FUNCTION_BLOCK fbV2_MainStationProcess

(*************************************************************** Ver.B1 - fbV2_StnSeqProcess - 161101 **************************************************************]

 	- Add 'bEffTimePriorityEn' to cutoff the process once effective time reached.																	
	- Change naming from 'bProcessCompleteBasedMasterTime' to 'bMinMaxEn'. 
	- 	
	- 
[****************************************************************************************************************************************************************************************************)

VAR_INPUT
	(*fbStnSeqProcess*)
	bAutoStartPbEn									: BOOL;
	bSavePB_Uni 									: BOOL; 														(*Universal*) (* Input - HMI - Save Push Button on Touchscreen*)
	bLoadPB_Uni 									: BOOL;														(*Universal*) (* Input - HMI - Load Push Button on Touchscreen*)
	bClearPB_SSER									: BOOL;
	bClearPB_SSUR									: BOOL;
	bTrackerEn										: BOOL;														(*During Tracker, it will only call arm when process completed*)
	bTrackerBasedOnPreviousTime					: BOOL;
	bMinMaxEn(*bProcessCompleteBasedMasterTime*)		: BOOL;
	bEffTimePriorityEn									: BOOL;
	bBasketTransferCallArmInterlock			: BOOL; (* Temporary -> for GPM Only*)

	(*fbGnrStationMasterController*)
	iCurrentStationAddress_Fix 							: INT;															(*Individual*) (* Input - Define current station no so that this fb know which array number to used*)
	iPreCallArmTime_Uni								: INT;															(*Universal*) (* Input - Pre-Call Arm Time, Program will call arm if the Total process timeEV Equal or Lesser than this value*)
	ARbAlternateStnEn								: ARRAY [1..iAlternateSetQty] OF BOOL;
	AR2siAlternateStn 									: ARRAY [1..iAlternateSetQty, 1..iAlternateStnQty] OF INT;

	
	
END_VAR

VAR_IN_OUT PERSISTENT

	(*fbStnSeqProcess*)
(*	DsStnSeqProInput_Ind 						: DS_StnSeqProInput;												(*Individual*) (* Input - PV of Instrument (Temperature, pressure, vacuum and etc), Signal of Sensor to allowed program under the current station status.*)
*)	DSStnSeqProcessCtrl_Ind			 		: DS_fbStnSeqProcessCtrl;											(*Individual*) (* InOut - Link with fbStnSeqProcess, so that this fb know the full status of fbStnSeqProcess and determine which action to take*)

	DsStnSeqRepStore_Ind 					: DSV2_fbStationSequenceRecipeStore; 								(*Individual*) (* InOut - HMI - The full set of DataStructure-StationSequenceRecipe should selectively display on HMI so that user can customise the recipe by choosing/configure the parameters.*)
	DsStnSubRepStore_Ind 					: DS_fbStationSubRecipeStore; 										(*Individual*) (* InOut - HMI - The full set of DataStructure-StationSubRecipe should selectively display on HMI so that user can customise the recipe by choosing/configure the parameters.*)
	DsStnSeqRepCall_Ind 						: DSV2_fbStationSequenceRecipeCall;									(*Individual*) (* InOut - Used to call StationSequenceRecipe Detail from fbStationSequenceRecipe*)
	DsStnSubRepCall_Ind 						: DS_fbStationSubRecipeCall;										(*Individual*) (* InOut - Used to call StationSubRecipe Detail from fbStationSubRecipe*)
	ARDsSSERSourceMinMaxTime_Uni						: ARRAY [1..iStnQty] OF DSV2_SSERSourceMinMaxTime;

	(*fbGnrStationMasterController*)
	ARbProductRecipeCallEn_Uni 				: ARRAY [0..iStnQty] OF BOOL;										(*Universal*) (* Output - Link with fbGnrProductRecipeMemory, Array based on Current Station No, the fbGnrProductRecipeMemory will start Read info from Memory when this bool turn on*)
	ARiProductRecipeNoCall_Uni 				: ARRAY [0..iStnQty] OF INT;										(*Universal*) (* Output - Link with fbGnrProductRecipeMemory, Array based on Current Station No, the read out from fbGnrProductRecipeMemory is based on this Product Recipe No*)
	ARiProductRecipeStepCall_Uni 				: ARRAY [0..iStnQty] OF INT;										(*Universal*) (* Output - Link with fbGnrProductRecipeMemory, Array based on Current Station No, the read out from fbGnrProductRecipeMemory is based on this Product Recipe Step No*)

	DSfbGnrProductRecipeMemoryOut_Uni 		: DSV2_fbGnrProductRecipeMemoryOut;								(*Universal*) (* Input - Link with fbGnrProductRecipeMemory, all the read out info from fbGnrProductRecipeMemory will store in this DataStucture*)

	ARbArmReady_Uni						: ARRAY [1..iArmQty] OF BOOL;										(* Universal*) (* Input  - From ArmPnpFB, This signal is used to confirm if the arm is ready and idling*)

	ARiStnNoToCalledArm_Uni					: ARRAY [0..iArmQty] OF INT; 										(*Universal*) (* Output - Link with fbArmPnP, Array based on Arm No, The Int will store which Station that calling the Arm*)
	ARDSGnrFeedArmPnpParameter_Uni		: ARRAY [0..iArmQty] OF DSV2_Gnr_CalledArmPnpParameter; 			(*Universal*) (* Output - Link with fbArmPnP, Array based on Current Station No, Arm should move based on this DataStructure Info*)

	ARDSLdBasketInfo_Uni		 			: ARRAY [0..iLdStnQty] OF DSV2_BasketInfo;								(*Input - Loading CONFIRM Basket Info*)
	ARDSUldBasketInfo_Uni		 			: ARRAY [0..iUldStnQty] OF DSV2_BasketInfo;							(*Input - Uloading CONFIRM Basket Info*)
	ARDsStnBasketInfo_Uni					: ARRAY [0..iStnQty] OF DSV2_BasketInfo;								(*Input - Station Basket Info*)



END_VAR

VAR_OUTPUT PERSISTENT
	bSaveInd_Uni 								: BOOL; 														(*Universal*) (* Output - HMI - Save Indicator on Touchscreen*)
	bLoadInd_Uni 								: BOOL; 														(*Universal*) (* Output - HMI - Load Indicator on Touchscreen*)
	bClearInd_SSER 								: BOOL;
	bClearInd_SSUR 								: BOOL;
(*	DSStnSeqProOutput_Ind 						:DS_StnSeqProOutput;											(*Individual*) (* Output - To Control Output - When process running, instrument should control by the output in this Data structure*)
*)

	bStationProcessCompleted : BOOL;
END_VAR



VAR PERSISTENT
	(*fbStnSeqProcess*)
	StnSeqProcessfb						: fbV2_StnSeqProcess;
	bStnSeqProcessStartInterlock			: BOOL;																	(*Individual*) (* Input - Interlocking to Enable the StnSeqProcess Start Signal, It might used on those station with Sliding door for close confirmation before process start*)

	(*fbGnrStationMasterController*)
	GnrStationMasterControllerfb				: fbV2_GnrStationMasterController;
	bStnSeqProcessSt						: BOOL;																(* Output - Link with fbStnSeqProcess, After Read out from fbGnrProductRecipeMemory, this fb will trigger this Bool to start the StnSeqProcess*)
	DSGnrBufferCalledArmPnpParameter 		: DSV2_Gnr_CalledArmPnpParameter;									(* Internal used, Buffer Data Structure read out from fbGnrProductRecipeMemory*)
	DSGnrBuffersPnpSequenceDescription		: STRING (99);														(* Internal used, Buffer Description read out from fbGnrProductRecipeMemory*)
	ARiPreviousStnSeqTotalProcessTime 		: ARRAY [0..iProductRecipeArrayQty] OF INT;								(* Internal used, Previous Total Process Time will save into this Array, Array based on StationSequenceNo*)
	iCallStep									: INT;																(* Internal used, to monitor the current Step so that you can indentify the error of this function block if stucked*)
	DSBasketInfo_Ind 							: DSV2_BasketInfo;														(*Individual*) (* InOut - Basket Information that comes into current station*)
	iNonStopCurrentProcessTime: INT;
END_VAR
VAR
	bLdStnConfirm: BOOL;
	bUldStnConfirm: BOOL;
	bStn1Confirm: BOOL;
	bGreaterStn1Confirm: BOOL;
	bLesserStnQtyConfirm: BOOL;
	bEqualStnQtyConfirm: BOOL;
	iTotalProcessTimeSV: INT;
	fbV2BasketInfoFinder_Ind: fbV2_BasketInfoFinder;
	iTotalProcessTimeCallForGnrStationMC: INT;
	iMasterTimeCallArmCountDownTime: INT;
	iMasterTimeBasedProcessCompleteFlag : BOOL;


	iMasterTimeBasedProcessCompleteFlagHR: BOOL;
	iProductRecipeBuffer: INT;
	bProductRecipeNoChangedFlag: BOOL;
END_VAR
VAR // added by the converter: edge detectors and wires of the graphical bodies
    _w1, _w2 : INT;
END_VAR

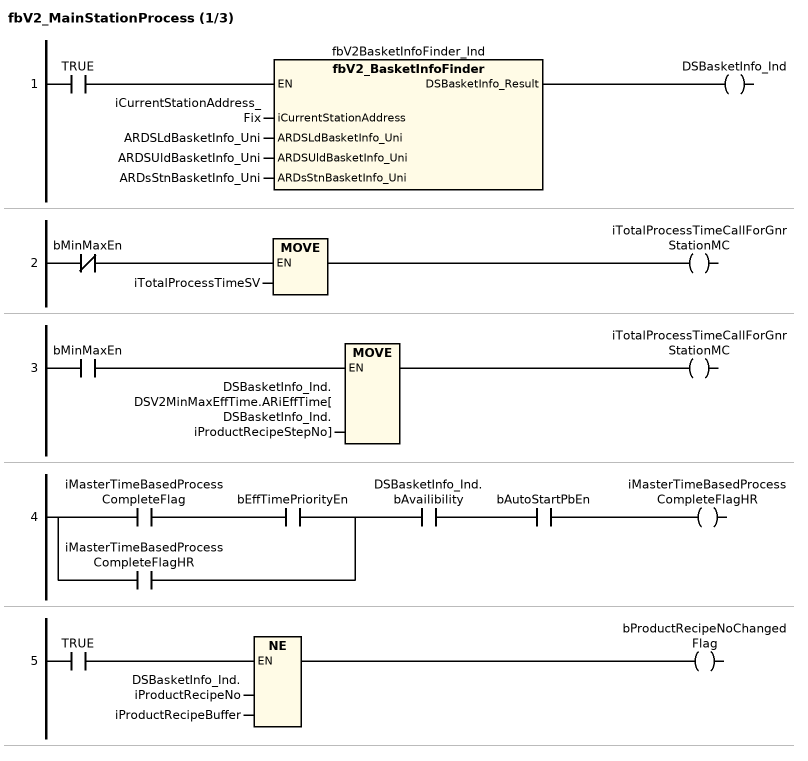
// NETWORK 1
fbV2BasketInfoFinder_Ind(
    iCurrentStationAddress := iCurrentStationAddress_Fix,
    ARDSLdBasketInfo_Uni := ARDSLdBasketInfo_Uni,
    ARDSUldBasketInfo_Uni := ARDSUldBasketInfo_Uni,
    ARDsStnBasketInfo_Uni := ARDsStnBasketInfo_Uni); // fbV2_BasketInfoFinder
DSBasketInfo_Ind := fbV2BasketInfoFinder_Ind.DSBasketInfo_Result;

// NETWORK 2
IF NOT bMinMaxEn THEN _w1 := iTotalProcessTimeSV; END_IF
iTotalProcessTimeCallForGnrStationMC := _w1;

// NETWORK 3
IF bMinMaxEn THEN
    _w2 := DSBasketInfo_Ind.DSV2MinMaxEffTime.ARiEffTime[DSBasketInfo_Ind.iProductRecipeStepNo];
END_IF
iTotalProcessTimeCallForGnrStationMC := _w2;

// NETWORK 4
iMasterTimeBasedProcessCompleteFlagHR := (iMasterTimeBasedProcessCompleteFlag AND bEffTimePriorityEn OR iMasterTimeBasedProcessCompleteFlagHR) AND DSBasketInfo_Ind.bAvailibility AND bAutoStartPbEn;

// NETWORK 5
bProductRecipeNoChangedFlag := DSBasketInfo_Ind.iProductRecipeNo <> iProductRecipeBuffer;

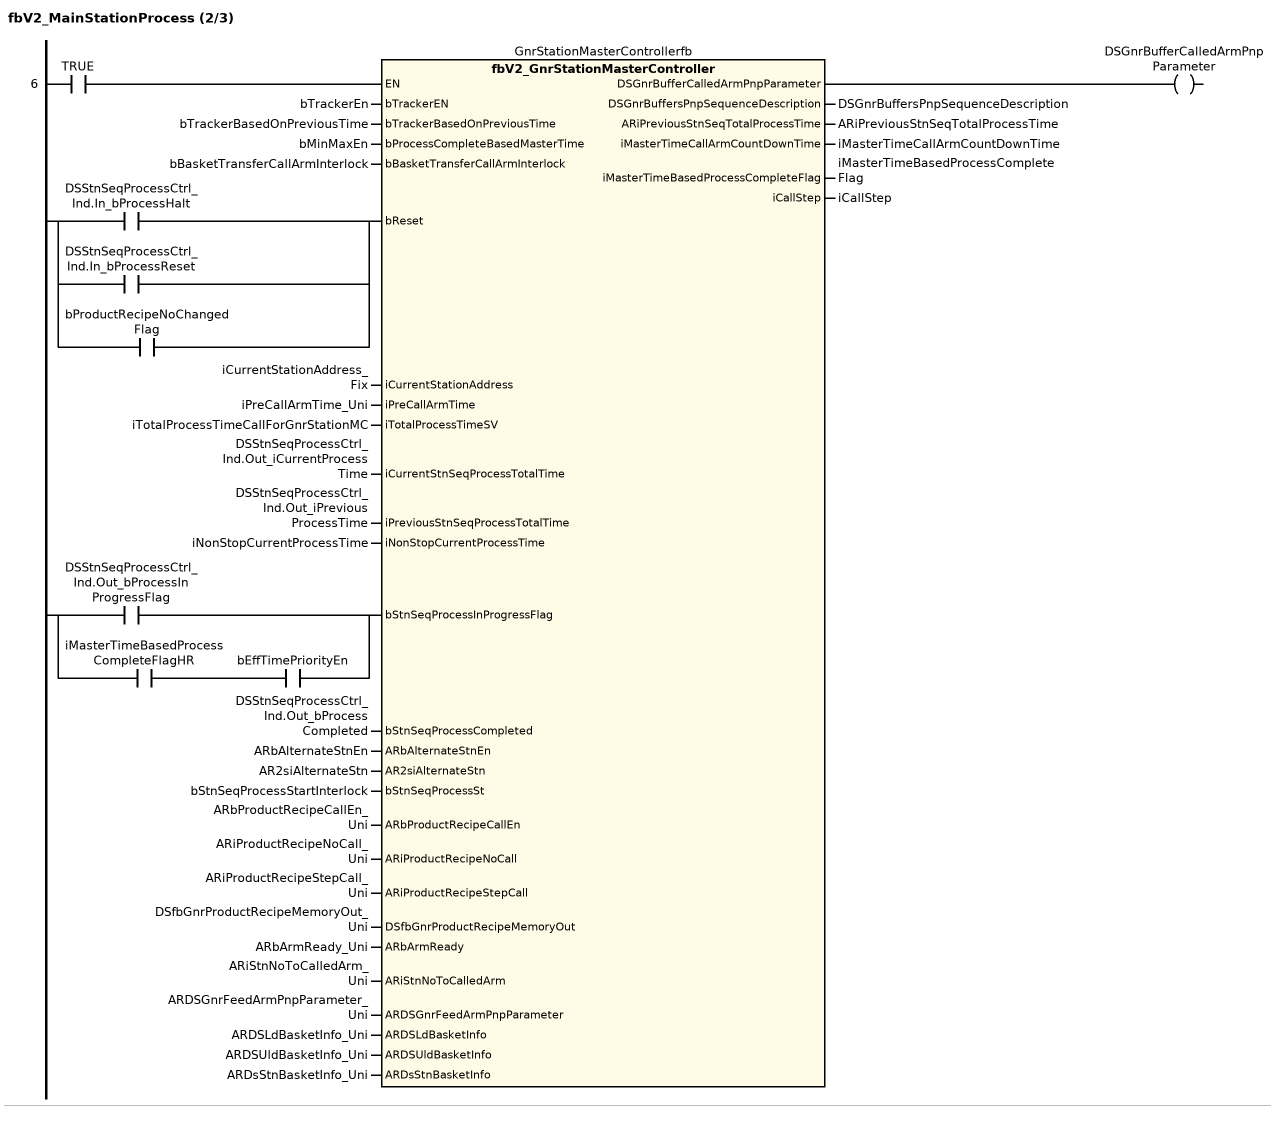
// NETWORK 6
GnrStationMasterControllerfb(
    bTrackerEN := bTrackerEn,
    bTrackerBasedOnPreviousTime := bTrackerBasedOnPreviousTime,
    bProcessCompleteBasedMasterTime := bMinMaxEn,
    bBasketTransferCallArmInterlock := bBasketTransferCallArmInterlock,
    bReset := DSStnSeqProcessCtrl_Ind.In_bProcessHalt OR DSStnSeqProcessCtrl_Ind.In_bProcessReset OR bProductRecipeNoChangedFlag,
    iCurrentStationAddress := iCurrentStationAddress_Fix,
    iPreCallArmTime := iPreCallArmTime_Uni,
    iTotalProcessTimeSV := iTotalProcessTimeCallForGnrStationMC,
    iCurrentStnSeqProcessTotalTime := DSStnSeqProcessCtrl_Ind.Out_iCurrentProcessTime,
    iPreviousStnSeqProcessTotalTime := DSStnSeqProcessCtrl_Ind.Out_iPreviousProcessTime,
    iNonStopCurrentProcessTime := iNonStopCurrentProcessTime,
    bStnSeqProcessInProgressFlag := DSStnSeqProcessCtrl_Ind.Out_bProcessInProgressFlag OR iMasterTimeBasedProcessCompleteFlagHR AND bEffTimePriorityEn,
    bStnSeqProcessCompleted := DSStnSeqProcessCtrl_Ind.Out_bProcessCompleted,
    ARbAlternateStnEn := ARbAlternateStnEn,
    AR2siAlternateStn := AR2siAlternateStn,
    bStnSeqProcessSt := bStnSeqProcessStartInterlock,
    ARbProductRecipeCallEn := ARbProductRecipeCallEn_Uni,
    ARiProductRecipeNoCall := ARiProductRecipeNoCall_Uni,
    ARiProductRecipeStepCall := ARiProductRecipeStepCall_Uni,
    DSfbGnrProductRecipeMemoryOut := DSfbGnrProductRecipeMemoryOut_Uni,
    ARbArmReady := ARbArmReady_Uni,
    ARiStnNoToCalledArm := ARiStnNoToCalledArm_Uni,
    ARDSGnrFeedArmPnpParameter := ARDSGnrFeedArmPnpParameter_Uni,
    ARDSLdBasketInfo := ARDSLdBasketInfo_Uni,
    ARDSUldBasketInfo := ARDSUldBasketInfo_Uni,
    ARDsStnBasketInfo := ARDsStnBasketInfo_Uni,
    DSGnrBuffersPnpSequenceDescription => DSGnrBuffersPnpSequenceDescription,
    ARiPreviousStnSeqTotalProcessTime => ARiPreviousStnSeqTotalProcessTime,
    iMasterTimeCallArmCountDownTime => iMasterTimeCallArmCountDownTime,
    iMasterTimeBasedProcessCompleteFlag => iMasterTimeBasedProcessCompleteFlag,
    iCallStep => iCallStep); // fbV2_GnrStationMasterController
DSGnrBufferCalledArmPnpParameter := GnrStationMasterControllerfb.DSGnrBufferCalledArmPnpParameter;

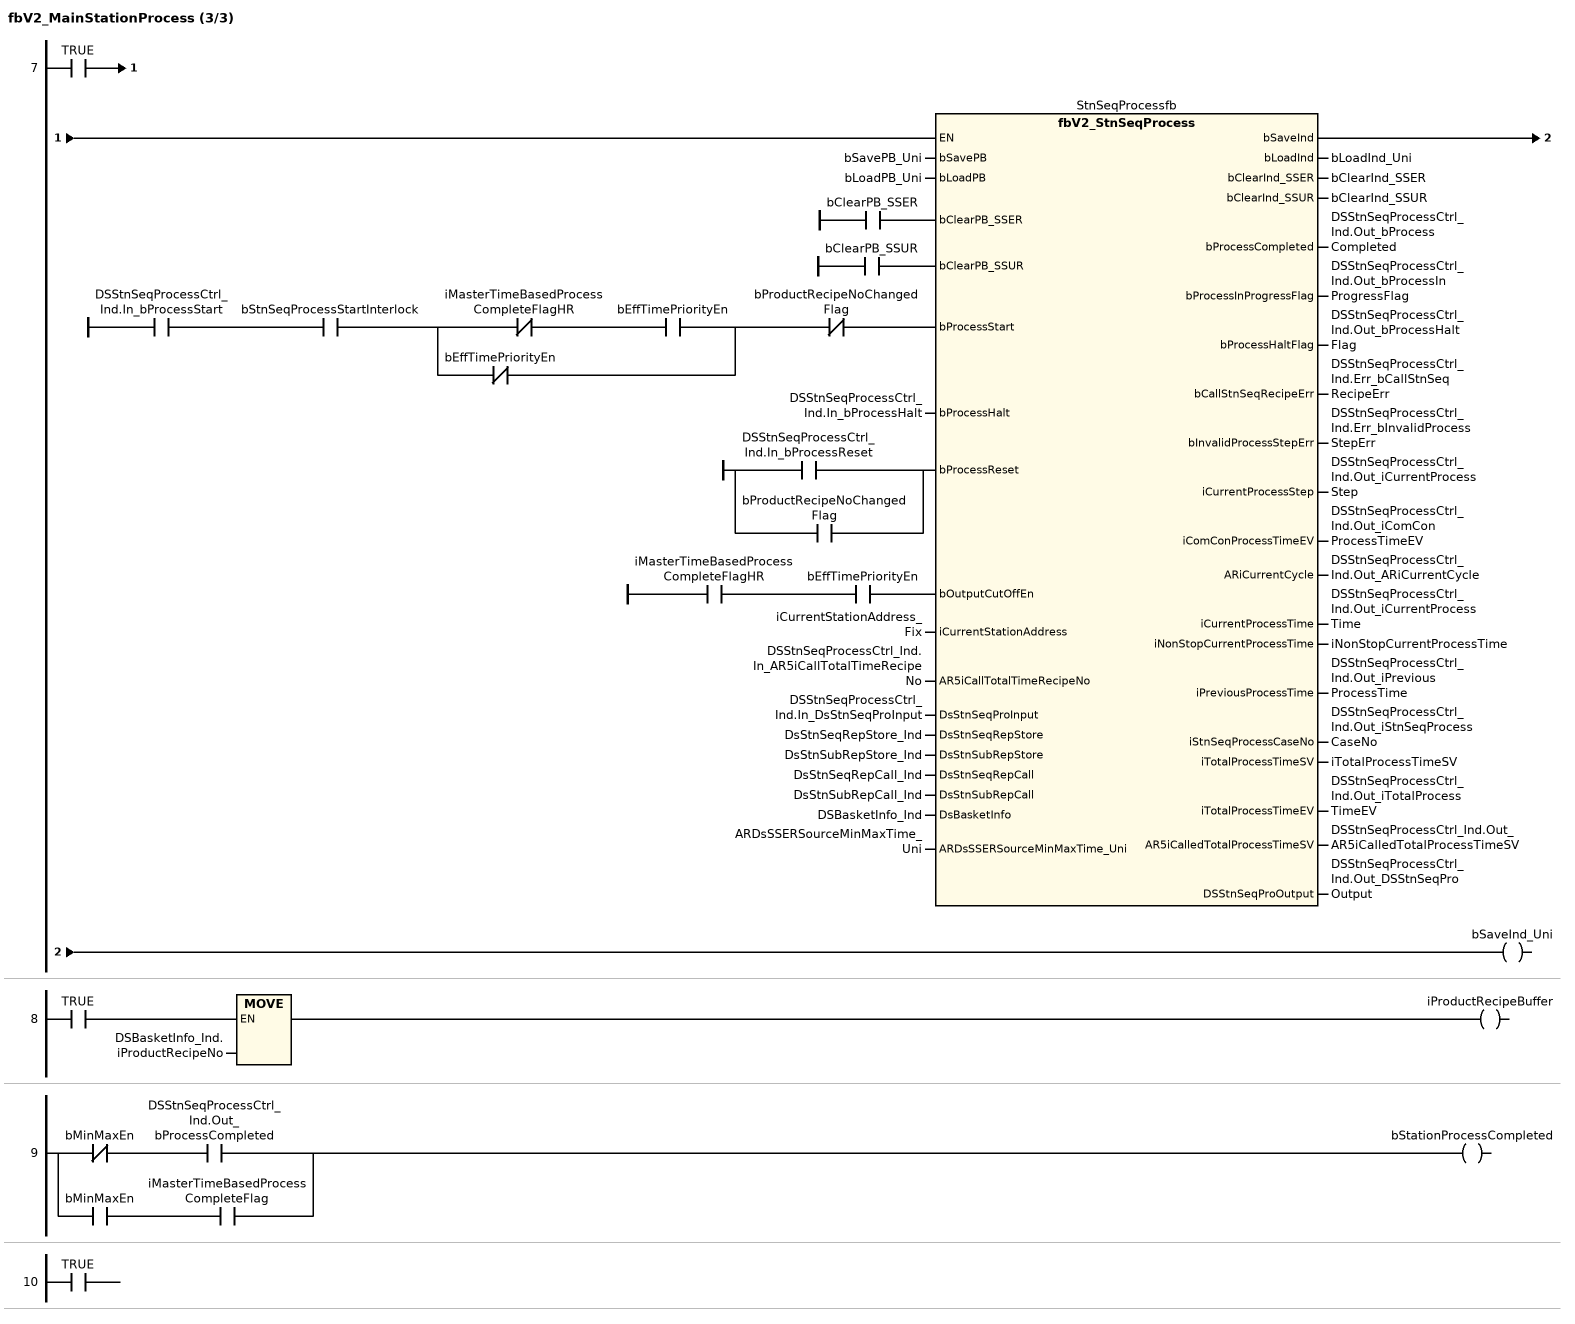
// NETWORK 7
StnSeqProcessfb(
    bSavePB := bSavePB_Uni,
    bLoadPB := bLoadPB_Uni,
    bClearPB_SSER := bClearPB_SSER,
    bClearPB_SSUR := bClearPB_SSUR,
    bProcessStart := ((DSStnSeqProcessCtrl_Ind.In_bProcessStart AND bStnSeqProcessStartInterlock) AND (NOT iMasterTimeBasedProcessCompleteFlagHR AND bEffTimePriorityEn OR NOT bEffTimePriorityEn)) AND NOT bProductRecipeNoChangedFlag,
    bProcessHalt := DSStnSeqProcessCtrl_Ind.In_bProcessHalt,
    bProcessReset := DSStnSeqProcessCtrl_Ind.In_bProcessReset OR bProductRecipeNoChangedFlag,
    bOutputCutOffEn := iMasterTimeBasedProcessCompleteFlagHR AND bEffTimePriorityEn,
    iCurrentStationAddress := iCurrentStationAddress_Fix,
    AR5iCallTotalTimeRecipeNo := DSStnSeqProcessCtrl_Ind.In_AR5iCallTotalTimeRecipeNo,
    DsStnSeqProInput := DSStnSeqProcessCtrl_Ind.In_DsStnSeqProInput,
    DsStnSeqRepStore := DsStnSeqRepStore_Ind,
    DsStnSubRepStore := DsStnSubRepStore_Ind,
    DsStnSeqRepCall := DsStnSeqRepCall_Ind,
    DsStnSubRepCall := DsStnSubRepCall_Ind,
    DsBasketInfo := DSBasketInfo_Ind,
    ARDsSSERSourceMinMaxTime_Uni := ARDsSSERSourceMinMaxTime_Uni,
    bLoadInd => bLoadInd_Uni,
    bClearInd_SSER => bClearInd_SSER,
    bClearInd_SSUR => bClearInd_SSUR,
    bProcessCompleted => DSStnSeqProcessCtrl_Ind.Out_bProcessCompleted,
    bProcessInProgressFlag => DSStnSeqProcessCtrl_Ind.Out_bProcessInProgressFlag,
    bProcessHaltFlag => DSStnSeqProcessCtrl_Ind.Out_bProcessHaltFlag,
    bCallStnSeqRecipeErr => DSStnSeqProcessCtrl_Ind.Err_bCallStnSeqRecipeErr,
    bInvalidProcessStepErr => DSStnSeqProcessCtrl_Ind.Err_bInvalidProcessStepErr,
    iCurrentProcessStep => DSStnSeqProcessCtrl_Ind.Out_iCurrentProcessStep,
    iComConProcessTimeEV => DSStnSeqProcessCtrl_Ind.Out_iComConProcessTimeEV,
    ARiCurrentCycle => DSStnSeqProcessCtrl_Ind.Out_ARiCurrentCycle,
    iCurrentProcessTime => DSStnSeqProcessCtrl_Ind.Out_iCurrentProcessTime,
    iNonStopCurrentProcessTime => iNonStopCurrentProcessTime,
    iPreviousProcessTime => DSStnSeqProcessCtrl_Ind.Out_iPreviousProcessTime,
    iStnSeqProcessCaseNo => DSStnSeqProcessCtrl_Ind.Out_iStnSeqProcessCaseNo,
    iTotalProcessTimeSV => iTotalProcessTimeSV,
    iTotalProcessTimeEV => DSStnSeqProcessCtrl_Ind.Out_iTotalProcessTimeEV,
    AR5iCalledTotalProcessTimeSV => DSStnSeqProcessCtrl_Ind.Out_AR5iCalledTotalProcessTimeSV,
    DSStnSeqProOutput => DSStnSeqProcessCtrl_Ind.Out_DSStnSeqProOutput); // fbV2_StnSeqProcess
bSaveInd_Uni := StnSeqProcessfb.bSaveInd;

// NETWORK 8
iProductRecipeBuffer := DSBasketInfo_Ind.iProductRecipeNo;

// NETWORK 9
bStationProcessCompleted := NOT bMinMaxEn AND DSStnSeqProcessCtrl_Ind.Out_bProcessCompleted OR bMinMaxEn AND iMasterTimeBasedProcessCompleteFlag;

// NETWORK 10

END_FUNCTION_BLOCK

(* stored: Version 1.1.0.1, ProductVersion 3.1.4024.12
   POU fbV2_MainStationProcess: Id {e9041466-6dcf-4c15-958a-c072fbce56a7}, SpecialFunc None *)
